{attribute 'linkalways'} 
{attribute 'no_explicit_call' := 'This FB is a CLASS and must be accessed using methods or properties'}
{attribute 'enable_dynamic_creation'}
FUNCTION_BLOCK FINAL NE_USINT EXTENDS Node
VAR
	in1 : _USINT(0);
	in2 : _USINT(0);
	out : _BOOL(FALSE);
END_VAR

METHOD PUBLIC Clone : I_Node
VAR
	pNode : POINTER TO NE_USINT;
END_VAR
pNode := __NEW(NE_USINT);
Clone := pNode^;
END_METHOD

METHOD FB_init : BOOL
VAR_INPUT
	bInitRetains : BOOL; // if TRUE, the retain variables are initialized (warm start / cold start)
	bInCopyCode : BOOL;  // if TRUE, the instance afterwards gets moved into the copy code (online change)
END_VAR
AddInput('in1',THIS^.in1);
AddInput('in2',THIS^.in2);
AddOutput('out', THIS^.out);
END_METHOD

METHOD PROTECTED OnExecute
VAR
END_VAR
out.Value := in1.Value <> in2.Value;
END_METHOD

END_FUNCTION_BLOCK

(* stored: Version 1.1.0.1, ProductVersion 3.1.4024.15
   POU NE_USINT: Id {7f8a9b89-ab7c-49ea-96eb-fe0c9f721dd3}, SpecialFunc None
   Folder Constructor: Id {da7f9b31-c8d0-4a4a-9b31-b728f6b5b723}
   Method Clone: Id {fee8917b-7a33-448f-8375-74868bba380f}
   Method FB_init: Id {96b661b4-59d9-4c7c-91de-938fb39ca0b5}
   Method OnExecute: Id {fedf7cb5-0aac-4120-9bbc-946ad0bc596a} *)
